(* CODESYS project ATV320_EL6751.library
   Author: 3threes
   Placeholder: ATV320
   Title: ATV320
   Version: 0.0.0.2
   DefaultNamespace: threesSoup01_ATV320
   Company: threesSoup01

Project tree, tasks and I/O mapping:
  libraries: Tc2_Standard, * (Beckhoff Automation GmbH); Tc2_System, * (Beckhoff Automation GmbH); Tc3_Module, * (Beckhoff Automation GmbH); VisuDialogs, * (System); VisuSymbols, 3.5.10.0 (System)
  DUTs/
    data type DUT_ATV320_Basic_HMI
    data type DUT_ATV320_Basic_HMI_PB
    data type DUT_ATV320_Basic_HMI_PL
    data type DUT_ATV320_NC1_CMD
    data type DUT_ATV320_NW1_ETA
    data type e_ATV320_OperationState
    interface ITF_ATV320_Basic: METH_CmdDisableOperation, METH_CmdDisableVoltage, METH_CmdEnableOperation, METH_CmdFaultReset, METH_CmdQuickStop, METH_CmdShutDown, METH_DriveRun, METH_Hz2RPM, METH_RPM2Hz, METH_SwitchOn, Prop_MaxHz, Prop_MaxRPM, Prop_NW1, Prop_OperationState
    data type u_ATV320_NC1_CMD
    data type u_ATV320_NW1_ETA
  GVLs/
    global variables GVL
  POUs/
    function block FB_ATV320_Basic [ST]: METH_CmdDisableOperation, METH_CmdDisableVoltage, METH_CmdEnableOperation, METH_CmdFaultReset, METH_CmdQuickStop, METH_CmdShutDown, METH_DriveRun, METH_Hz2RPM, METH_RPM2Hz, METH_SwitchOn, Prop_MaxHz, Prop_MaxRPM, Prop_NW1, Prop_OperationState
    function block FB_ATV320_Basic_withHMI [ST]: METH_HMIUpdate
  Version/
    global variables Global_Version
  VISUs/
    visualisation Visualization
  text list GlobalTextList
*)

// DUTs/DUT_ATV320_Basic_HMI
TYPE DUT_ATV320_Basic_HMI :
STRUCT
	PB			:DUT_ATV320_Basic_HMI_PB;
	PL			:DUT_ATV320_Basic_HMI_PL;
END_STRUCT
END_TYPE

// DUTs/DUT_ATV320_Basic_HMI_PB
TYPE DUT_ATV320_Basic_HMI_PB :
STRUCT
	bReset					:BOOL;
	bEnableOperation		:BOOL;
	bSwitchON				:BOOL;
	bDriveRun				:BOOL;
	bDisableOperation		:BOOL;
	bDisableVoltage			:BOOL;
	bQuickStop				:BOOL;
	bShutdown				:BOOL;
	iSetPoint				:INT;
END_STRUCT
END_TYPE

// DUTs/DUT_ATV320_Basic_HMI_PL
TYPE DUT_ATV320_Basic_HMI_PL :
STRUCT
	rCurrentHz		:REAL;
	rCurrentRPM		:REAL;
	State			:e_ATV320_OperationState;
END_STRUCT
END_TYPE

// DUTs/DUT_ATV320_NC1_CMD
TYPE DUT_ATV320_NC1_CMD :
STRUCT
	b00SwitchON				:BIT;
	b01EnableVoltage		:BIT;
	b02QuickStop			:BIT;
	b03EnableOperation		:BIT;
	b04,b05,b06				:BIT;	//Reserved
	b07FaultReset			:BIT;
	b08Halt					:BIT;
	b09,b10					:BIT;	//Reserved
	b11,b12,b13,b14,b15		:BIT;	//Manufacturer specific assignable
END_STRUCT
END_TYPE

// DUTs/DUT_ATV320_NW1_ETA
TYPE DUT_ATV320_NW1_ETA :
STRUCT
	b00Ready2SwitchON			:BIT;
	b01SwitchON					:BIT;
	b02OperationEnabled			:BIT;
	b03Fault					:BIT;
	b04VoltageEnabled			:BIT;
	b05QuickStopped				:BIT;
	b06SwitchONDisabled			:BIT;
	b07Warning					:BIT;
	b08							:BIT;
	b09Remote					:BIT;
	b10TargetReached			:BIT;
	b11InternalLimitActive		:BIT;
	b12,b13						:BIT;
	b14StopKeyFromManufacturer	:BIT;
	b15DriectionFromManufacturer:BIT;
	
END_STRUCT
END_TYPE

// DUTs/e_ATV320_OperationState
{attribute 'qualified_only'}
{attribute 'strict'}
TYPE e_ATV320_OperationState :
(
	None					:=0
	,NoReady2SwitchOn 		:=1
	,Switched2Disabled		:=2
	,Ready2SwitchOn			:=3
	,SwitchedOn				:=4
	,OperationEnabled		:=5
	,QuickStoppedActivate	:=6
	,FauleReactionActivate	:=7
	,Fault					:=8
);
END_TYPE

// DUTs/u_ATV320_NC1_CMD
TYPE u_ATV320_NC1_CMD :
UNION
	raw				:UINT;
	CMD				:DUT_ATV320_NC1_CMD;
END_UNION
END_TYPE

// DUTs/u_ATV320_NW1_ETA
TYPE u_ATV320_NW1_ETA :
UNION
	raw				:UINT;
	ETA				:DUT_ATV320_NW1_ETA;
END_UNION
END_TYPE

// GVLs/GVL
{attribute 'qualified_only'}
VAR_GLOBAL
	Device1_From0State AT %I*:UINT;
	StatusWord   at %i*:uint;
END_VAR

// Version/Global_Version
{attribute 'TcGenerated'}
{attribute 'no-analysis'}
{attribute 'linkalways'}
// This function has been automatically generated from the project information.
VAR_GLOBAL CONSTANT
	{attribute 'const_non_replaced'}
	stLibVersion_ATV320 : ST_LibVersion := (iMajor := 0, iMinor := 0, iBuild := 0, iRevision := 2, nFlags := 0, sVersion := '0.0.0.2');
END_VAR

// DUTs/ITF_ATV320_Basic
INTERFACE ITF_ATV320_Basic

METHOD METH_CmdDisableOperation : BOOL
VAR_INPUT
	iTrigger	:Bool;
END_VAR
END_METHOD

METHOD METH_CmdDisableVoltage : BOOL
VAR_INPUT
	iTrigger	:Bool;
END_VAR
END_METHOD

METHOD METH_CmdEnableOperation : BOOL
VAR_INPUT
	iTrigger	:Bool;
END_VAR
END_METHOD

METHOD METH_CmdFaultReset : BOOL
VAR_INPUT
	iTrigger:BOOL;
END_VAR
END_METHOD

METHOD METH_CmdQuickStop : BOOL
VAR_INPUT
	iTrigger	:Bool;
END_VAR
END_METHOD

METHOD METH_CmdShutDown : BOOL
VAR_INPUT
	iTrigger	:Bool;
END_VAR
END_METHOD

METHOD METH_DriveRun : BOOL
VAR_INPUT
	iTrigger	:BOOL;
	iSetPoint	:int;
END_VAR
END_METHOD

METHOD METH_Hz2RPM : INT
VAR_INPUT
	iData		:REAL;
END_VAR
END_METHOD

METHOD METH_RPM2Hz : REAL
VAR_INPUT
	iData			:INT;
END_VAR
END_METHOD

METHOD METH_SwitchOn : BOOL
VAR_INPUT
	iTrigger:BOOL;
END_VAR
END_METHOD

PROPERTY Prop_MaxHz : Real
GET
END_GET
SET
END_SET
END_PROPERTY

PROPERTY Prop_MaxRPM : Real
GET
END_GET
SET
END_SET
END_PROPERTY

PROPERTY Prop_NW1 : UINT
GET
END_GET
END_PROPERTY

PROPERTY Prop_OperationState : e_ATV320_OperationState
GET
END_GET
END_PROPERTY

END_INTERFACE

// POUs/FB_ATV320_Basic
FUNCTION_BLOCK PUBLIC FB_ATV320_Basic IMPLEMENTS ITF_ATV320_Basic
VAR_INPUT
END_VAR
VAR_OUTPUT
END_VAR
VAR
	_OperationState		:e_ATV320_OperationState;
	_MaxHz				:REAL:=50.0;
	_MaxRPM				:REAL:=1500.0;
END_VAR

//Process IO
	VAR
		//INPUTS
			NW1			AT%I*		:u_ATV320_NW1_ETA;
			NW2			AT%I*		:INT;
		//OUTPUTs
			NC1			AT%Q*		:u_ATV320_NC1_CMD;
			NC2			AT%Q*		:INT;
	END_VAR

VAR CONSTANT
	_c_ETAMask			:WORD:=16#006F;
END_VAR

METHOD METH_CmdDisableOperation : BOOL
VAR_INPUT
	iTrigger	: BOOL;
END_VAR

METH_CmdDisableOperation:=FALSE;
IF iTrigger THEN
	NC1.CMD.b03EnableOperation:=FALSE;
	METH_CmdDisableOperation:= TRUE;
	NC2:=0;
END_IF

;
END_METHOD

METHOD METH_CmdDisableVoltage : BOOL
VAR_INPUT
	iTrigger	: BOOL;
END_VAR
METH_CmdDisableVoltage:=FALSE;
IF iTrigger THEN
	NC1.raw:=16#0;
	METH_CmdDisableVoltage:=TRUE;
	NC2:=0;
;
END_IF
END_METHOD

METHOD METH_CmdEnableOperation : BOOL
VAR_INPUT
	iTrigger	: BOOL;
END_VAR

NC1.CMD.b03EnableOperation:=iTrigger 
AND (Prop_OperationState = e_ATV320_OperationState.SwitchedOn
OR Prop_OperationState = e_ATV320_OperationState.OperationEnabled);
;
END_METHOD

METHOD METH_CmdFaultReset : BOOL
VAR_INPUT
	iTrigger	: BOOL;
END_VAR

METH_CmdFaultReset:=FALSE;
NC1.CMD.b07FaultReset:= Prop_OperationState = e_ATV320_OperationState.Fault AND iTrigger;
IF NC1.CMD.b07FaultReset THEN
	METH_CmdFaultReset:=TRUE;
	NC2:=0;
END_IF;
END_METHOD

METHOD METH_CmdQuickStop : BOOL
VAR_INPUT
	iTrigger	: BOOL;
END_VAR
IF iTrigger THEN
	NC1.raw:=16#02;
	NC2:=0;
;
END_IF

METH_CmdDisableVoltage(Prop_OperationState = e_ATV320_OperationState.QuickStoppedActivate);

METH_CmdQuickStop:=Prop_OperationState = e_ATV320_OperationState.Switched2Disabled;
END_METHOD

METHOD METH_CmdShutDown : BOOL
VAR_INPUT
	iTrigger	: BOOL;
END_VAR
METH_CmdShutDown:=FALSE;
IF iTrigger THEN
	NC1.raw:=16#06;
	METH_CmdShutDown:=TRUE;
	NC2:=0;
END_IF
END_METHOD

METHOD METH_DriveRun : BOOL
VAR_INPUT
	iTrigger	: BOOL;
	iSetPoint	: INT;
END_VAR

IF iTrigger AND Prop_OperationState = e_ATV320_OperationState.OperationEnabled THEN
	NC2:= iSetPoint;
END_IF
END_METHOD

METHOD METH_Hz2RPM : INT
VAR_INPUT
	iData	: REAL;
END_VAR

METH_Hz2RPM:=
REAL_TO_INT(
(iData/_MaxHz)*_MaxRPM)
;
END_METHOD

METHOD METH_RPM2Hz : REAL
VAR_INPUT
	iData	: INT;
END_VAR
METH_RPM2Hz:=

INT_TO_REAL(iData)/_MaxRPM*_MaxHz;
END_METHOD

METHOD METH_SwitchOn : BOOL
VAR_INPUT
	iTrigger	: BOOL;
END_VAR
VAR_INST
	R_TRIG		:R_TRIG;
	TON			:TON;
	State		:e_ATV320_OperationState;
	Step			:INT;
END_VAR


TON.PT:=T#1S;
METH_SwitchOn:=FALSE;

R_TRIG(CLK:=iTrigger);

IF R_TRIG.Q THEN
	Step:=5;
END_IF


CASE Step OF
	
	5:
		NC1.CMD.b00SwitchON:=FALSE;
		NC1.CMD.b01EnableVoltage:=FALSE;
		NC1.CMD.b02QuickStop:=FALSE;
		TON(IN:=FALSE);
		Step:=10;

	10:
		NC1.CMD.b01EnableVoltage:=TRUE;
		NC1.CMD.b02QuickStop:=TRUE;
		Step:=15;
	15:
		TON(
			IN:=NOT Prop_OperationState = e_ATV320_OperationState.Ready2SwitchOn
			);
		IF TON.Q THEN
			Step:=999;
		END_IF
		IF Prop_OperationState = e_ATV320_OperationState.Ready2SwitchOn THEN
			TON(IN:=FALSE);
			Step:=20;
		END_IF
	20:
		NC1.CMD.b00SwitchON:=TRUE;
		Step:=25;
	25:
		NC1.CMD.b00SwitchON:=TRUE;
		TON(
			IN:=NOT Prop_OperationState = e_ATV320_OperationState.SwitchedOn
			);
		IF TON.Q THEN
			Step:=999;
		END_IF
		IF Prop_OperationState = e_ATV320_OperationState.SwitchedOn THEN
			Step:=30;
			TON(IN:=FALSE);
		END_IF
	30:
		NC1.CMD.b03EnableOperation:=TRUE;
		Step:=40;
	40:
		NC1.CMD.b03EnableOperation:=TRUE;
		TON(
			IN:=NOT Prop_OperationState = e_ATV320_OperationState.OperationEnabled
			);
		IF TON.Q THEN
			Step:=999;
		END_IF
		IF Prop_OperationState = e_ATV320_OperationState.OperationEnabled THEN
			Step:=50;
			TON(IN:=FALSE);
		END_IF
	50:
		METH_SwitchOn:=TRUE;

	999:
		NC1.CMD.b00SwitchON:=FALSE;
		NC1.CMD.b01EnableVoltage:=FALSE;
		NC1.CMD.b02QuickStop:=FALSE;
		NC1.CMD.b03EnableOperation:=FALSE;
		Step:=0;
		
END_CASE
END_METHOD

PROPERTY Prop_MaxHz : REAL
GET
Prop_MaxHz:=_MaxHz;
END_GET
SET


_MaxHz:=Prop_MaxHz;
END_SET
END_PROPERTY

{warning 'add property implementation'}
PROPERTY Prop_MaxRPM : REAL
GET
Prop_MaxRPM:=_MaxRPM;
END_GET
SET
_MaxRPM:=Prop_MaxRPM;
END_SET
END_PROPERTY

{warning 'add property implementation'}
PROPERTY Prop_NW1 : UINT
GET
Prop_NW1:=NW1.raw;
END_GET
END_PROPERTY

{warning 'add property implementation'}
PROPERTY Prop_OperationState : e_ATV320_OperationState
GET
VAR
	StateAfterMasked		:UINT;
END_VAR

StateAfterMasked:=Prop_NW1 AND _c_ETAMask;

//Init
Prop_OperationState:=e_ATV320_OperationState.NoReady2SwitchOn;

CASE StateAfterMasked OF
	
	16#0040:
		Prop_OperationState:=e_ATV320_OperationState.Switched2Disabled;
		
	16#0021:
		Prop_OperationState:=e_ATV320_OperationState.Ready2SwitchOn;
		
	16#0023:
		Prop_OperationState:=e_ATV320_OperationState.SwitchedOn;
		
	16#0027:
		Prop_OperationState:=e_ATV320_OperationState.OperationEnabled;
		
	16#0007:
		Prop_OperationState:=e_ATV320_OperationState.QuickStoppedActivate;
		
	16#002F:
		Prop_OperationState:=e_ATV320_OperationState.FauleReactionActivate;
		
	16#0008,16#0028:
		Prop_OperationState:=e_ATV320_OperationState.Fault;


END_CASE
END_GET
END_PROPERTY

END_FUNCTION_BLOCK

// POUs/FB_ATV320_Basic_withHMI
FUNCTION_BLOCK FB_ATV320_Basic_withHMI EXTENDS FB_ATV320_Basic
VAR_INPUT
END_VAR
VAR_OUTPUT
END_VAR
VAR
	_HMI			:DUT_ATV320_Basic_HMI;
END_VAR

METHOD PUBLIC METH_HMIUpdate : BOOL


METH_CmdFaultReset(iTrigger:=_HMI.PB.bReset);
METH_SwitchOn(iTrigger:=_HMI.PB.bSwitchON);
METH_DriveRun(
	iTrigger:=Prop_OperationState = e_ATV320_OperationState.OperationEnabled
	,iSetPoint:=_HMI.PB.iSetPoint
);
METH_CmdDisableOperation(iTrigger:=_HMI.PB.bDisableOperation);
METH_CmdDisableVoltage(iTrigger:=_HMI.PB.bDisableVoltage);
METH_CmdQuickStop(iTrigger:=_HMI.PB.bQuickStop);
METH_CmdShutDown(iTrigger:=_HMI.PB.bShutdown);

_HMI.PL.rCurrentHz:=METH_RPM2Hz(iData:=NW2);
_HMI.PL.rCurrentRPM:=NW2;
_HMI.PL.State:=Prop_OperationState;
END_METHOD

END_FUNCTION_BLOCK

// VISUs/Visualization
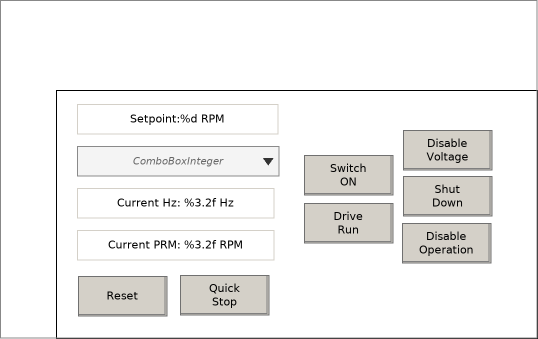
VISUALIZATION Visualization  // 538x339
VAR_IN_OUT
	HMI			:DUT_ATV320_Basic_HMI;
END_VAR
    RoundedRectangle (56,90 482x249)
    Button (402,223 89x40), "Disable Operation"
        tap HMI.PB.bDisableOperation
    Button (403,130 89x40), "Disable Voltage"
        tap HMI.PB.bDisableVoltage
    Button (304,203 89x40), "Drive Run"
        tap HMI.PB.bDriveRun
    Button (180,275 89x40), "Quick Stop"
        tap HMI.PB.bReset
    Button (78,276 89x40), "Reset"
        tap HMI.PB.bReset
    Button (403,176 89x40), "Shut Down"
        tap HMI.PB.bShutdown
    Button (304,155 89x40), "Switch ON"
        tap HMI.PB.bSwitchON
    Textfield (77,104 201x30), "Setpoint:%d RPM", text variable: HMI.PB.iSetPoint
        OnMouseClick: write the text variable via VisuDialogs.Numpad
    ComboBoxInteger (77,146 202x30), variable: HMI.PL.State, input disabled if: TRUE
    Textfield (77,188 197x30), "Current Hz: %3.2f Hz", text variable: HMI.PL.rCurrentHz
    Textfield (77,230 197x30), "Current PRM: %3.2f RPM", text variable: HMI.PL.rCurrentRPM
END_VISUALIZATION
